(* checks a string for various characteristics and returns a string if validation fails *)
FUNCTION F_ValidateString : T_MaxString
VAR_INPUT
	strFieldData		: T_MaxString;	(* string to be examined *)
	nExpectedChars		: BYTE;			(* >0 = no of chars expected in string, 0 = chars not counted but string must not be empty *)
	nMaxChars			: UINT;			(* >0 = max no of chars allowed in strFieldData, 0 = do not check *)
	bNumCharsOnly		: BOOL;			(* TRUE = all chars are checked to ensure only numerical (0-9) chars are present *)
	bDecPointAllowed	: BOOL;			(* TRUE = decimal point is allowed in a numerical string *)
END_VAR
VAR
	nIndex				: INT;
	nCharValue			: BYTE;
END_VAR
(*
-------------------------------------------------------------------------------------------------
DATE		Version	Author	Comments
-------------------------------------------------------------------------------------------------
30/01/2015	3.00.00	PB		Initial release

-------------------------------------------------------------------------------------------------
*)

(* string contains data *)
IF LEN(strFieldData) > 0 THEN

	(* field data length exceeds specified maximum no of chars *)
	IF nMaxChars > 0 AND LEN(strFieldData) >= nMaxChars THEN

		F_ValidateString := 'XML field data contains too many chars';

	(* string has expected no of chars OR string length does not matter *)
	ELSIF LEN(strFieldData) = nExpectedChars OR nExpectedChars = 0 THEN

		(* string must only have numerical chars *)
		IF bNumCharsOnly = TRUE THEN

			(* check each char in the string *)
			FOR nIndex := 1 TO LEN(strFieldData) DO

				(* convert char to ASCII value *)
				nCharValue := F_ToASC(MID(strFieldData, 1, nIndex));

				(* string char is valid if 0-9, decimal point also allowed if enabled *)
				IF (nCharValue >= F_ToASC('0') AND nCharValue <= F_ToASC('9')) OR (nCharValue = F_ToASC('.') AND bDecPointAllowed = TRUE) THEN

					F_ValidateString := '';

				(* invalid char *)
				ELSE

					F_ValidateString := F_CONCAT3('Invalid char "', MID(strFieldData, 1, nIndex), '" found');
					EXIT;
				END_IF
			END_FOR

		(* string can be alpha-numeric chars *)
		ELSE

			F_ValidateString := '';
		END_IF

	(* string has incorrect no of chars *)
	ELSE

		F_ValidateString := F_CONCAT4('Expected length = ', BYTE_TO_STRING(nExpectedChars), ', actual length = ', INT_TO_STRING(LEN(strFieldData)));
	END_IF

(* empty string *)
ELSE

	F_ValidateString := 'Empty';
END_IF

END_FUNCTION

(* stored: Version 1.1.0.1, ProductVersion 3.1.4024.15
   POU F_ValidateString: Id {67445dd5-d33f-4ae7-b075-e2003487029b}, SpecialFunc None *)
